(* Schneider Machine Expert - Basic project SAU1, file version 2.0.0.0 *)
(* ProjectInformations: Name=New project *)

HARDWARE
  Cpu 0: TM221CE16T
  Cartridge1 0: TMC2SL1
  EthernetConfiguration: NetworkName=M221, IpAllocationMode=FixedAddress, IpAddress=192.168.1.11, SubnetMask=255.255.255.0
  EthernetConfiguration: NetworkName=M221, IpAllocationMode=FixedAddress, IpAddress=0.0.0.0, SubnetMask=0.0.0.0
  SerialLineConfiguration: Baud=Baud9600, Parity=ParityNone, DataBits=DataBits8, StopBits=StopBits1, PhysicalMedium=PhysicalMediumRs485, TransmissionMode=TransmissionModeModbusRtu, SlaveId=1, Addressing=MasterAddressing
  MastTask: UsePeriodScanMode=false, PeriodScan=100
  FastTask: Period=255
  CpuBehavior: StartingMode=StartAsPreviousState, AutoSaveRamOnEeprom=true, WatchdogPeriod=250

SYMBOLS  (address, symbol, comment, settings)
  %S5       SB_TB100MS  "内部时钟生成的 100 毫秒时基"
  %TM0        [Preset=15, Base=OneSecond]
  %TM1        [Preset=10, Base=TenMilliSeconds]
  %TM2        [Preset=15, Base=OneSecond]
  %TM3        [Preset=15, Base=OneSecond]
  %TM4        [Preset=15, Base=OneSecond]
  %READ_VAR0   [Link(Value(FBComLinkParameterEnums=SerialLine1)), RemoteDeviceId(Value(int=1)), Timeout(Value(int=3)), ObjType(Value(FBComObjTypeParameterEnums=IW)), FirstObj(Value(int=513)), Quantity(Value(int=4)), IndexData(Value(int=0))]
  %READ_VAR1   [Link(Value(FBComLinkParameterEnums=SerialLine1)), RemoteDeviceId(Value(int=3)), Timeout(Value(int=3)), ObjType(Value(FBComObjTypeParameterEnums=IW)), FirstObj(Value(int=513)), Quantity(Value(int=11)), IndexData(Value(int=10))]
  %READ_VAR2   [Link(Value(FBComLinkParameterEnums=SerialLine1)), RemoteDeviceId(Value(int=2)), Timeout(Value(int=3)), ObjType(Value(FBComObjTypeParameterEnums=IW)), FirstObj(Value(int=513)), Quantity(Value(int=3)), IndexData(Value(int=5))]
  %READ_VAR3   [Link(Value(FBComLinkParameterEnums=SerialLine1)), RemoteDeviceId(Value(int=4)), Timeout(Value(int=3)), ObjType(Value(FBComObjTypeParameterEnums=IW)), FirstObj(Value(int=513)), Quantity(Value(int=8)), IndexData(Value(int=30))]
  %READ_VAR4   [Link(Value(FBComLinkParameterEnums=SerialLine1)), RemoteDeviceId(Value(int=3)), Timeout(Value(int=3)), ObjType(Value(FBComObjTypeParameterEnums=IW)), FirstObj(Value(int=536)), Quantity(Value(int=1)), IndexData(Value(int=25))]

POU Communication
  (* SectionNumber=0 *)

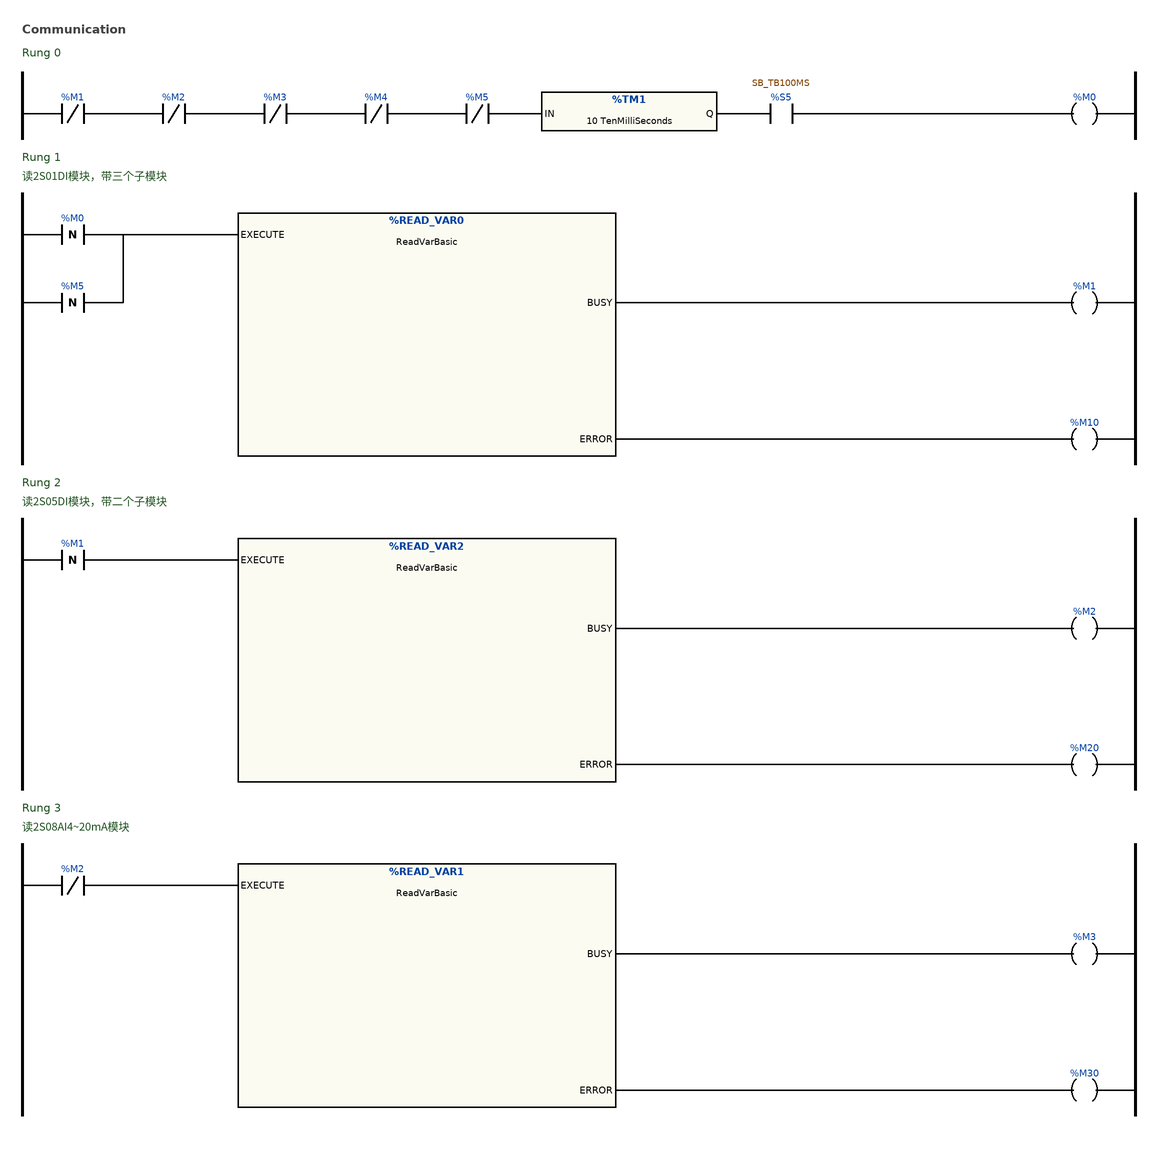

// Rung 0
  BLK %TM1
  LDN %M1
  ANDN %M2
  ANDN %M3
  ANDN %M4
  ANDN %M5
  IN
  OUT_BLK
  LD Q
  AND %S5                 (* SB_TB100MS *)
  ST %M0
  END_BLK
  // as ST:
  //   %TM1(IN := NOT %M1 AND NOT %M2 AND NOT %M3 AND NOT %M4 AND NOT %M5);
  //   %M0 := %TM1.Q AND SB_TB100MS;

// Rung 1
// 读2S01DI模块，带三个子模块
  BLK %READ_VAR0
  LDF %M0
  ORF %M5
  EXECUTE
  OUT_BLK
  LD BUSY
  ST %M1
  LD ERROR
  ST %M10
  END_BLK
  // as ST:
  //   %READ_VAR0(EXECUTE := FALLING(%M0) OR FALLING(%M5));
  //   %M1 := %READ_VAR0.BUSY;
  //   %M10 := %READ_VAR0.ERROR;

// Rung 2
// 读2S05DI模块，带二个子模块
  BLK %READ_VAR2
  LDF %M1
  EXECUTE
  OUT_BLK
  LD BUSY
  ST %M2
  LD ERROR
  ST %M20
  END_BLK
  // as ST:
  //   %READ_VAR2(EXECUTE := FALLING(%M1));
  //   %M2 := %READ_VAR2.BUSY;
  //   %M20 := %READ_VAR2.ERROR;

// Rung 3
// 读2S08AI4~20mA模块
  BLK %READ_VAR1
  LDN %M2
  EXECUTE
  OUT_BLK
  LD BUSY
  ST %M3
  LD ERROR
  ST %M30
  END_BLK
  // as ST:
  //   %READ_VAR1(EXECUTE := NOT %M2);
  //   %M3 := %READ_VAR1.BUSY;
  //   %M30 := %READ_VAR1.ERROR;

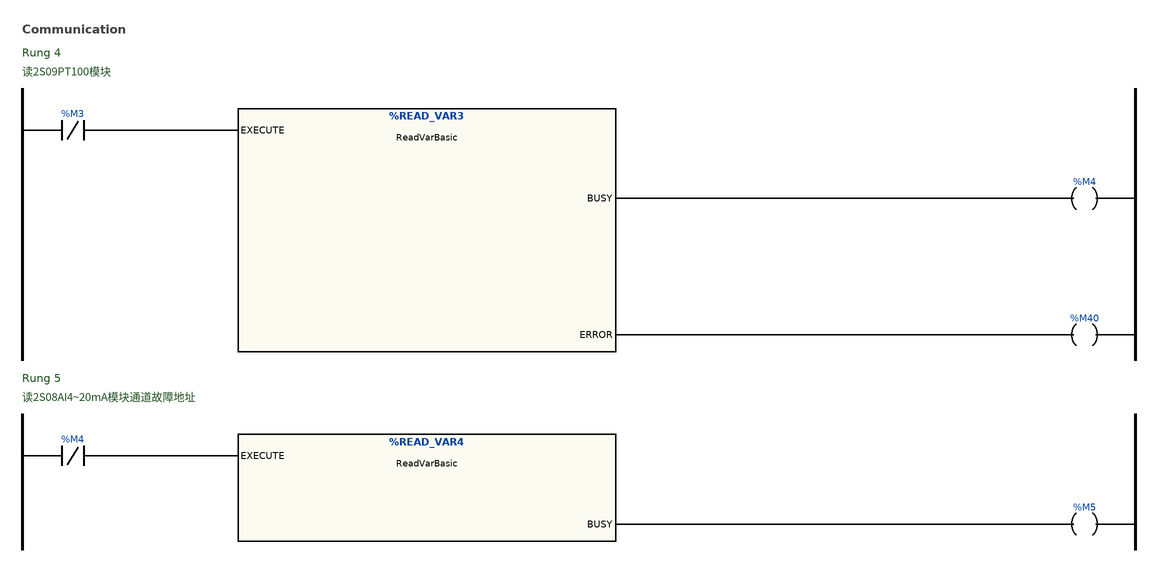

// Rung 4
// 读2S09PT100模块
  BLK %READ_VAR3
  LDN %M3
  EXECUTE
  OUT_BLK
  LD BUSY
  ST %M4
  LD ERROR
  ST %M40
  END_BLK
  // as ST:
  //   %READ_VAR3(EXECUTE := NOT %M3);
  //   %M4 := %READ_VAR3.BUSY;
  //   %M40 := %READ_VAR3.ERROR;

// Rung 5
// 读2S08AI4~20mA模块通道故障地址
  BLK %READ_VAR4
  LDN %M4
  EXECUTE
  OUT_BLK
  LD BUSY
  ST %M5
  END_BLK
  // as ST:
  //   %READ_VAR4(EXECUTE := NOT %M4);
  //   %M5 := %READ_VAR4.BUSY;

POU CommError
  (* SectionNumber=0 *)

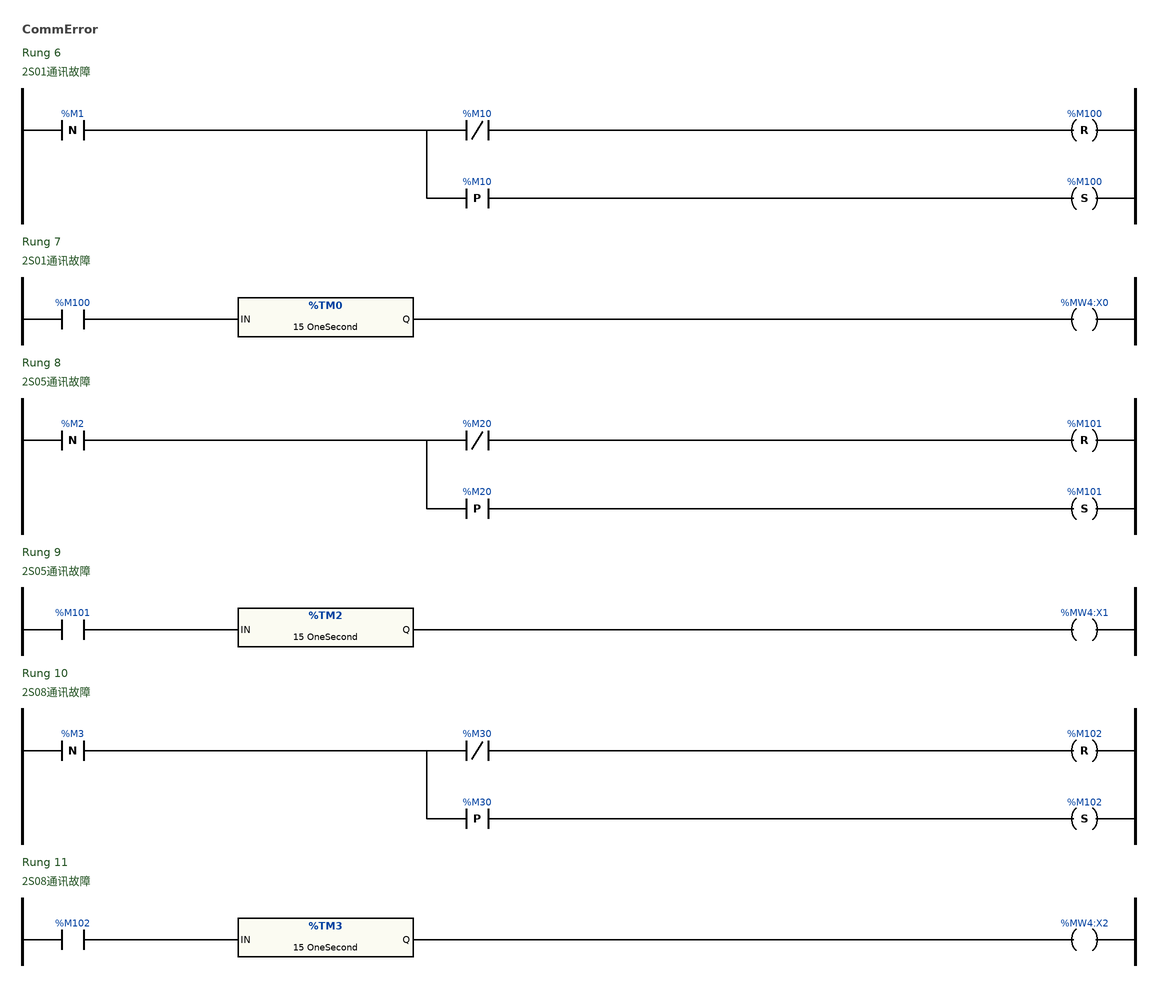

// Rung 6
// 2S01通讯故障
  LDF %M1
  MPS
  ANDN %M10
  R %M100
  MPP
  ANDR %M10
  S %M100
  // as ST:
  //   IF FALLING(%M1) AND NOT %M10 THEN %M100 := FALSE; END_IF;
  //   IF FALLING(%M1) AND RISING(%M10) THEN %M100 := TRUE; END_IF;

// Rung 7
// 2S01通讯故障
  BLK %TM0
  LD %M100
  IN
  OUT_BLK
  LD Q
  ST %MW4:X0
  END_BLK
  // as ST:
  //   %TM0(IN := %M100);
  //   %MW4:X0 := %TM0.Q;

// Rung 8
// 2S05通讯故障
  LDF %M2
  MPS
  ANDN %M20
  R %M101
  MPP
  ANDR %M20
  S %M101
  // as ST:
  //   IF FALLING(%M2) AND NOT %M20 THEN %M101 := FALSE; END_IF;
  //   IF FALLING(%M2) AND RISING(%M20) THEN %M101 := TRUE; END_IF;

// Rung 9
// 2S05通讯故障
  BLK %TM2
  LD %M101
  IN
  OUT_BLK
  LD Q
  ST %MW4:X1
  END_BLK
  // as ST:
  //   %TM2(IN := %M101);
  //   %MW4:X1 := %TM2.Q;

// Rung 10
// 2S08通讯故障
  LDF %M3
  MPS
  ANDN %M30
  R %M102
  MPP
  ANDR %M30
  S %M102
  // as ST:
  //   IF FALLING(%M3) AND NOT %M30 THEN %M102 := FALSE; END_IF;
  //   IF FALLING(%M3) AND RISING(%M30) THEN %M102 := TRUE; END_IF;

// Rung 11
// 2S08通讯故障
  BLK %TM3
  LD %M102
  IN
  OUT_BLK
  LD Q
  ST %MW4:X2
  END_BLK
  // as ST:
  //   %TM3(IN := %M102);
  //   %MW4:X2 := %TM3.Q;

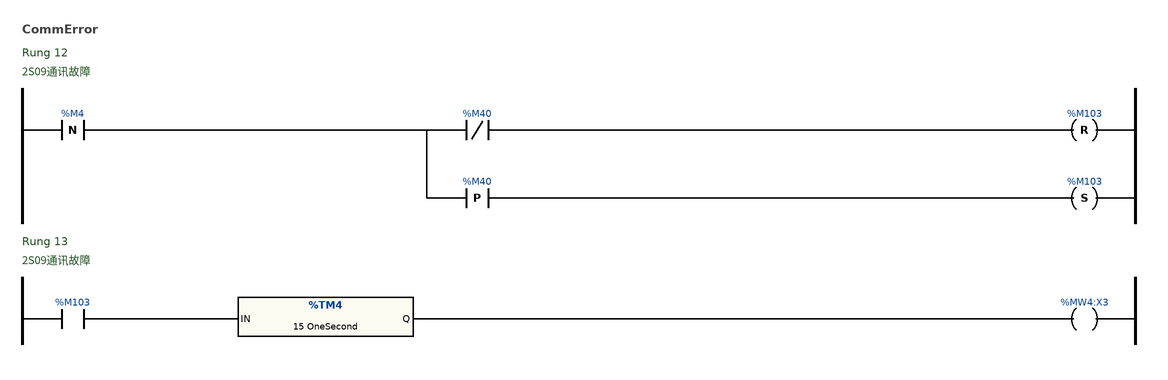

// Rung 12
// 2S09通讯故障
  LDF %M4
  MPS
  ANDN %M40
  R %M103
  MPP
  ANDR %M40
  S %M103
  // as ST:
  //   IF FALLING(%M4) AND NOT %M40 THEN %M103 := FALSE; END_IF;
  //   IF FALLING(%M4) AND RISING(%M40) THEN %M103 := TRUE; END_IF;

// Rung 13
// 2S09通讯故障
  BLK %TM4
  LD %M103
  IN
  OUT_BLK
  LD Q
  ST %MW4:X3
  END_BLK
  // as ST:
  //   %TM4(IN := %M103);
  //   %MW4:X3 := %TM4.Q;
